Staubli VAL3: convGetName.pgx

program convGetName(string& x_sFileName[] (dimensions=1))
begin
  // This program asks the user to enter a name for
  // a new conveyor calibration data file and
  // store it onto the flashdisk.
  //
  //
  // Created 23-02-05                                   C.CURRIVAND
  //----------------------------------------------------------------
  //
  call up:type(0,12,lang:sListOfMessage[21])
  call up:read(len(lang:sListOfMessage[21]),12,x_sFileName,8,false)
  call up:clear(0,12)
end
